TYPE E_ControlSource : (
    CONTROL_SOURCE_INVALID := 0,
    CONTROL_SOURCE_LOCAL := 10,
    CONTROL_SOURCE_ROBOT := 20
); END_TYPE

(* stored: Version 1.1.0.1
   DUT E_ControlSource: Id {E3000000-0000-4000-8000-000000000002} *)
